TYPE eParIDAccessState :
	(
		ParID_STATE_WAIT := 0,
		ParID_STATE_READY,
		ParID_STATE_READ_SDO,
		ParID_STATE_WRITE_SDO,		
		ParID_STATE_ERROR
	);
END_TYPE

(* stored: Version 1.1.0.1, ProductVersion 3.1.4024.3
   DUT eParIDAccessState: Id {3d63862b-5def-0e17-177d-631440498d8c} *)
